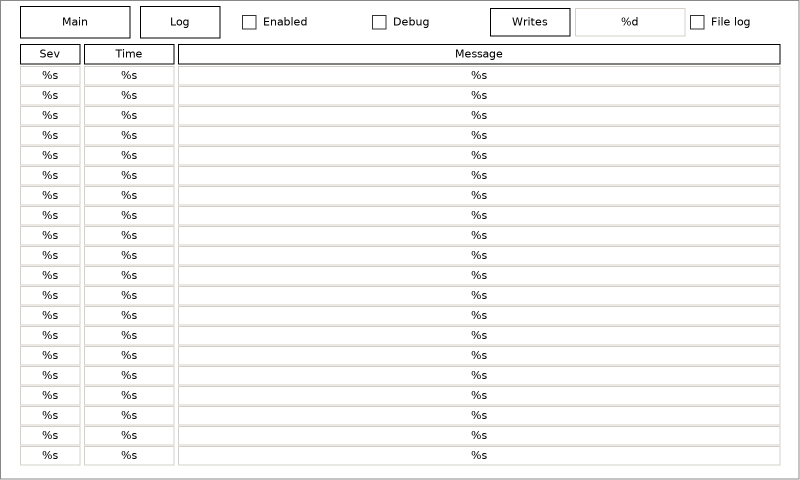
VISUALIZATION Logs  // 800x480
    Rectangle (20,6 110x32), "Main"
        OnMouseDown: change screen: Main
    Rectangle (140,6 80x32), "Log"
    Checkbox (240,8 120x28), "Enabled", variable: GVL_Log.bLogEnabled
    Checkbox (370,8 110x28), "Debug", variable: GVL_Log.bDebugMode
    Checkbox (688,8 110x28), "File log", variable: GVL_HmiPersistent.stLogFileCfg.bEnabled
    Rectangle (490,8 80x28), "Writes"
    Textfield (575,8 110x28), "%d", text variable: GVL_Log.nWriteIdx
    Rectangle (20,44 60x20), "Sev"
    Rectangle (84,44 90x20), "Time"
    Rectangle (178,44 602x20), "Message"
    Textfield (20,66 60x19), "%s", text variable: GVL_Log.aRecent[0].sSevText
    Textfield (84,66 90x19), "%s", text variable: GVL_Log.aRecent[0].sTime
    Textfield (178,66 602x19), "%s", text variable: GVL_Log.aRecent[0].sMsg
    Textfield (20,86 60x19), "%s", text variable: GVL_Log.aRecent[1].sSevText
    Textfield (84,86 90x19), "%s", text variable: GVL_Log.aRecent[1].sTime
    Textfield (178,86 602x19), "%s", text variable: GVL_Log.aRecent[1].sMsg
    Textfield (20,106 60x19), "%s", text variable: GVL_Log.aRecent[2].sSevText
    Textfield (84,106 90x19), "%s", text variable: GVL_Log.aRecent[2].sTime
    Textfield (178,106 602x19), "%s", text variable: GVL_Log.aRecent[2].sMsg
    Textfield (20,126 60x19), "%s", text variable: GVL_Log.aRecent[3].sSevText
    Textfield (84,126 90x19), "%s", text variable: GVL_Log.aRecent[3].sTime
    Textfield (178,126 602x19), "%s", text variable: GVL_Log.aRecent[3].sMsg
    Textfield (20,146 60x19), "%s", text variable: GVL_Log.aRecent[4].sSevText
    Textfield (84,146 90x19), "%s", text variable: GVL_Log.aRecent[4].sTime
    Textfield (178,146 602x19), "%s", text variable: GVL_Log.aRecent[4].sMsg
    Textfield (20,166 60x19), "%s", text variable: GVL_Log.aRecent[5].sSevText
    Textfield (84,166 90x19), "%s", text variable: GVL_Log.aRecent[5].sTime
    Textfield (178,166 602x19), "%s", text variable: GVL_Log.aRecent[5].sMsg
    Textfield (20,186 60x19), "%s", text variable: GVL_Log.aRecent[6].sSevText
    Textfield (84,186 90x19), "%s", text variable: GVL_Log.aRecent[6].sTime
    Textfield (178,186 602x19), "%s", text variable: GVL_Log.aRecent[6].sMsg
    Textfield (20,206 60x19), "%s", text variable: GVL_Log.aRecent[7].sSevText
    Textfield (84,206 90x19), "%s", text variable: GVL_Log.aRecent[7].sTime
    Textfield (178,206 602x19), "%s", text variable: GVL_Log.aRecent[7].sMsg
    Textfield (20,226 60x19), "%s", text variable: GVL_Log.aRecent[8].sSevText
    Textfield (84,226 90x19), "%s", text variable: GVL_Log.aRecent[8].sTime
    Textfield (178,226 602x19), "%s", text variable: GVL_Log.aRecent[8].sMsg
    Textfield (20,246 60x19), "%s", text variable: GVL_Log.aRecent[9].sSevText
    Textfield (84,246 90x19), "%s", text variable: GVL_Log.aRecent[9].sTime
    Textfield (178,246 602x19), "%s", text variable: GVL_Log.aRecent[9].sMsg
    Textfield (20,266 60x19), "%s", text variable: GVL_Log.aRecent[10].sSevText
    Textfield (84,266 90x19), "%s", text variable: GVL_Log.aRecent[10].sTime
    Textfield (178,266 602x19), "%s", text variable: GVL_Log.aRecent[10].sMsg
    Textfield (20,286 60x19), "%s", text variable: GVL_Log.aRecent[11].sSevText
    Textfield (84,286 90x19), "%s", text variable: GVL_Log.aRecent[11].sTime
    Textfield (178,286 602x19), "%s", text variable: GVL_Log.aRecent[11].sMsg
    Textfield (20,306 60x19), "%s", text variable: GVL_Log.aRecent[12].sSevText
    Textfield (84,306 90x19), "%s", text variable: GVL_Log.aRecent[12].sTime
    Textfield (178,306 602x19), "%s", text variable: GVL_Log.aRecent[12].sMsg
    Textfield (20,326 60x19), "%s", text variable: GVL_Log.aRecent[13].sSevText
    Textfield (84,326 90x19), "%s", text variable: GVL_Log.aRecent[13].sTime
    Textfield (178,326 602x19), "%s", text variable: GVL_Log.aRecent[13].sMsg
    Textfield (20,346 60x19), "%s", text variable: GVL_Log.aRecent[14].sSevText
    Textfield (84,346 90x19), "%s", text variable: GVL_Log.aRecent[14].sTime
    Textfield (178,346 602x19), "%s", text variable: GVL_Log.aRecent[14].sMsg
    Textfield (20,366 60x19), "%s", text variable: GVL_Log.aRecent[15].sSevText
    Textfield (84,366 90x19), "%s", text variable: GVL_Log.aRecent[15].sTime
    Textfield (178,366 602x19), "%s", text variable: GVL_Log.aRecent[15].sMsg
    Textfield (20,386 60x19), "%s", text variable: GVL_Log.aRecent[16].sSevText
    Textfield (84,386 90x19), "%s", text variable: GVL_Log.aRecent[16].sTime
    Textfield (178,386 602x19), "%s", text variable: GVL_Log.aRecent[16].sMsg
    Textfield (20,406 60x19), "%s", text variable: GVL_Log.aRecent[17].sSevText
    Textfield (84,406 90x19), "%s", text variable: GVL_Log.aRecent[17].sTime
    Textfield (178,406 602x19), "%s", text variable: GVL_Log.aRecent[17].sMsg
    Textfield (20,426 60x19), "%s", text variable: GVL_Log.aRecent[18].sSevText
    Textfield (84,426 90x19), "%s", text variable: GVL_Log.aRecent[18].sTime
    Textfield (178,426 602x19), "%s", text variable: GVL_Log.aRecent[18].sMsg
    Textfield (20,446 60x19), "%s", text variable: GVL_Log.aRecent[19].sSevText
    Textfield (84,446 90x19), "%s", text variable: GVL_Log.aRecent[19].sTime
    Textfield (178,446 602x19), "%s", text variable: GVL_Log.aRecent[19].sMsg
END_VISUALIZATION

(* stored: Version 1.1.0.1, ProductVersion 3.1.4024.16
   Visu Logs: Id {a1b2c3d4-0e5f-4a6b-9c7d-000000000103} *)
